FUNCTION_BLOCK FB_HMI
VAR_INPUT
END_VAR
VAR_OUTPUT
END_VAR
VAR
END_VAR

END_FUNCTION_BLOCK

(* stored: Version 1.1.0.1, ProductVersion 3.1.4024.10
   POU FB_HMI: Id {cafd80df-fe24-46eb-a55a-3bd2734d0ece}, SpecialFunc None *)
